ABB RAPID module: Wobj_base_Nest.mod

MODULE Wobj_base_Nest
	! Points are read in order of declaration.
  ! Please do not change the order of points!

  LOCAL PERS robtarget pWobj_U_PointX1:=[[1366.482,-44.35383,-437.2596],[0.00289803114719689,0.518160820007324,-0.855277180671692,0.00138014717958868],[-1,-1,-1,0],[9E+09,9E+09,9E+09,9E+09,9E+09,9E+09]];
	LOCAL PERS robtarget pWobj_U_PointX2:=[[499.4017,-779.6686,-454.657],[0.00289512774907053,0.51816987991333,-0.855271697044373,0.00139488652348518],[-1,-1,-2,0],[9E+09,9E+09,9E+09,9E+09,9E+09,9E+09]];
	LOCAL PERS robtarget pWobj_U_PointY1:=[[1787.532,-537.8456,-434.5679],[0.00288750068284571,0.518146634101868,-0.85528576374054,0.00139471667353064],[-1,-1,-1,0],[9E+09,9E+09,9E+09,9E+09,9E+09,9E+09]];

ENDMODULE
